SUBAPPLICATION RampLimitFS_TO_logiBUS_QDA_PWM_OPC (* Ein PWM-Kanal (0-100% Duty): VT-Zahlenfeld+Balkengrafik+6 Ramp-Tasten, physischer PWM-Ausgang, OPC-UA Publish/Subscribe (generisch, ein Kanal) *)
  (* Standard: 61499-2; Description: Copyright (c) 2026 Meisterschulen am Ostbahnhof This program and the accompanying materials are made available under the terms of the Eclipse Public License 2.0 which is available at https://www.eclipse.org/legal/epl-2.0/ SPDX-License-Identifier: EPL-2.0 *)
  (* Version 1.0, 2026-08-28, Franz Höpfinger, Meisterschulen am Ostbahnhof, initial API and implementation and/or initial documentation *)
  PACKAGE MyLib::sys;
  IMPORT isobus::UT::Q::const::IDs::ID_NULL;
  IMPORT logiBUS::io::DQ::logiBUS_DO;
  IMPORT logiBUS::io::DQ::logiBUS_DO_S;
  IMPORT isobus::UT::io::Button::ButtonActivationCode::BT_PRESSED_LATCHED;
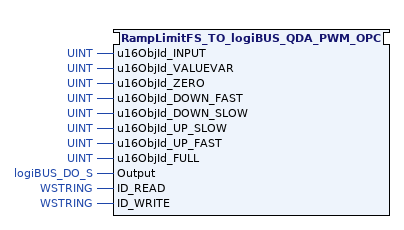
  VAR_INPUT
    u16ObjId_INPUT : UINT := ID_NULL; (* Object ID CInputNumber (Duty-Eingabe/-Anzeige, roh 0..64255 = 0.000-100.000%) *)
    u16ObjId_VALUEVAR : UINT := ID_NULL; (* Object ID CNumberVariable (Prozent 0-100, gemeinsam gebunden an Balkengrafik und CInputNumber-Anzeige) *)
    u16ObjId_ZERO : UINT := ID_NULL; (* Object ID Taste '0' (RampLimitFS.ZERO) *)
    u16ObjId_DOWN_FAST : UINT := ID_NULL; (* Object ID Taste '--' (RampLimitFS.DOWN_FAST, ~10%) *)
    u16ObjId_DOWN_SLOW : UINT := ID_NULL; (* Object ID Taste '-' (RampLimitFS.DOWN_SLOW, ~1%) *)
    u16ObjId_UP_SLOW : UINT := ID_NULL; (* Object ID Taste '+' (RampLimitFS.UP_SLOW, ~1%) *)
    u16ObjId_UP_FAST : UINT := ID_NULL; (* Object ID Taste '++' (RampLimitFS.UP_FAST, ~10%) *)
    u16ObjId_FULL : UINT := ID_NULL; (* Object ID Taste 'F' (RampLimitFS.FULL, 100%) *)
    Output : logiBUS::io::DQ::logiBUS_DO_S := logiBUS_DO::Invalid; (* Identify the PWM Output Output_Q1..Q12 *)
    ID_READ : WSTRING; (* Remote-Sollwert-Adresse (Prozent REAL, ACTION=SUBSCRIBE) *)
    ID_WRITE : WSTRING; (* Echo-Ruckmelde-Adresse (Prozent REAL, ACTION=PUBLISH) *)
  END_VAR
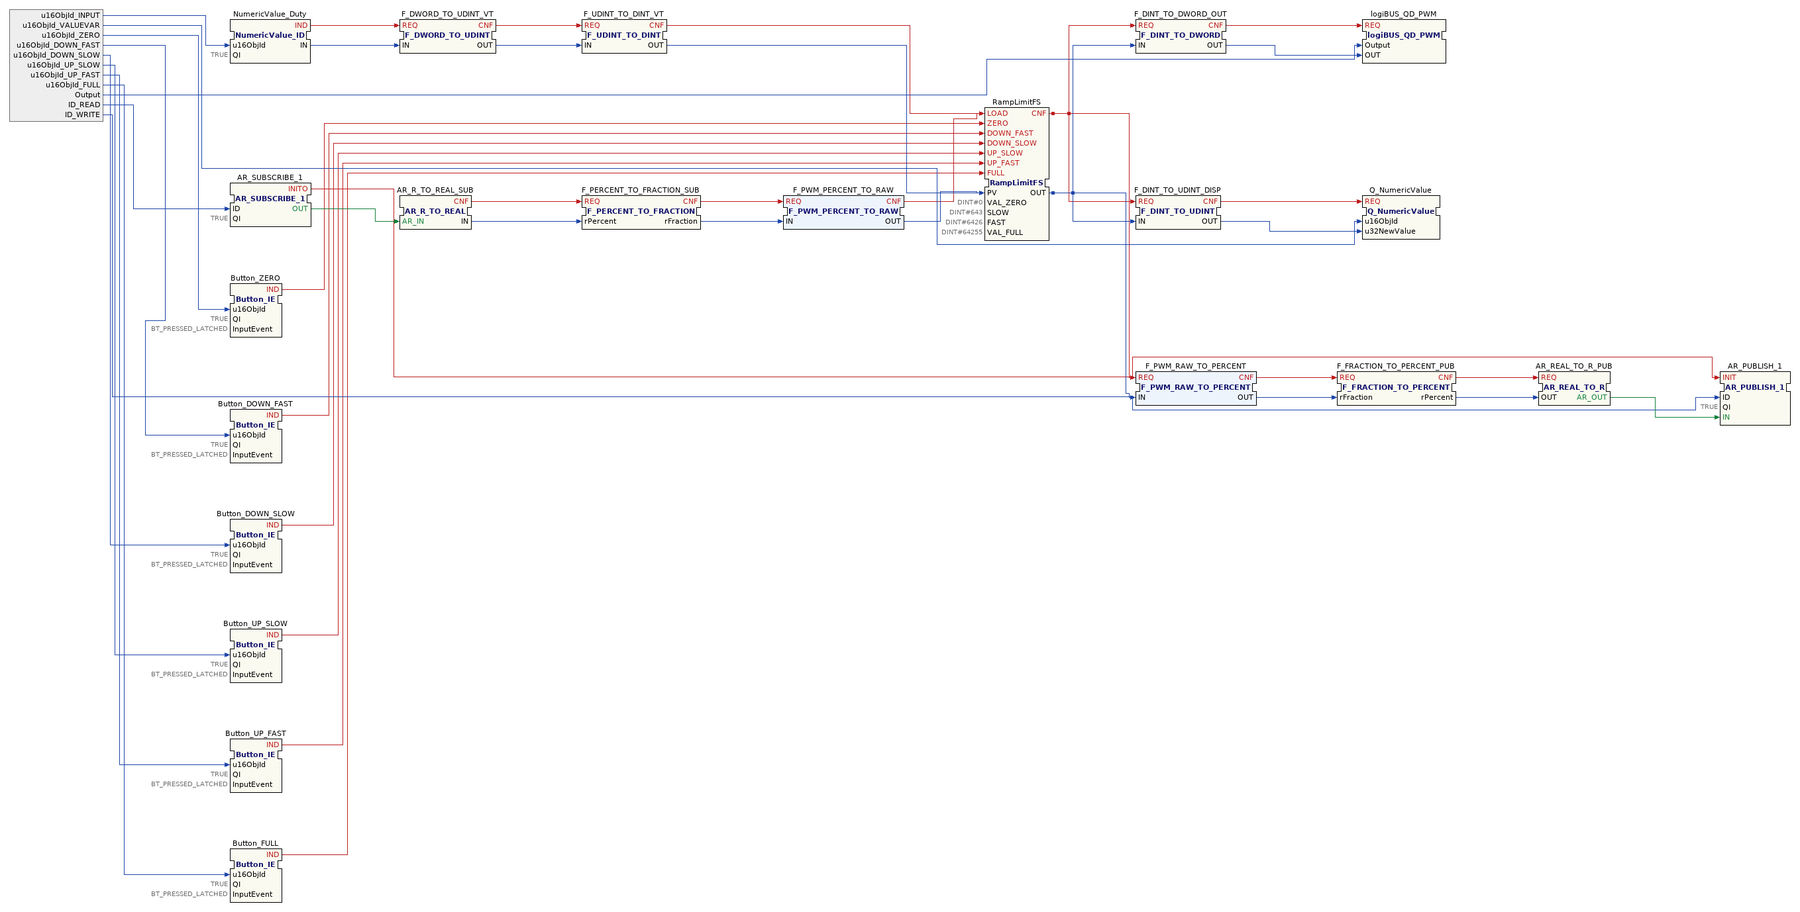
  FBS
    NumericValue_Duty : isobus::UT::io::NumericValue::NumericValue_ID(QI := TRUE);
    F_DWORD_TO_UDINT_VT : iec61131::conversion::F_DWORD_TO_UDINT;
    F_UDINT_TO_DINT_VT : iec61131::conversion::F_UDINT_TO_DINT;
    AR_SUBSCRIBE_1 : adapter::net::AR_SUBSCRIBE_1(QI := TRUE);
    AR_R_TO_REAL_SUB : adapter::conversion::unidirectional::AR_R_TO_REAL;
    F_PERCENT_TO_FRACTION_SUB : logiBUS::signalprocessing::fieldbus::F_PERCENT_TO_FRACTION;
    RampLimitFS : eclipse4diac::signalprocessing::RampLimitFS(VAL_ZERO := DINT#0, SLOW := DINT#643, FAST := DINT#6426, VAL_FULL := DINT#64255);
    Button_ZERO : isobus::UT::io::Button::Button_IE(QI := TRUE, InputEvent := BT_PRESSED_LATCHED);
    Button_DOWN_FAST : isobus::UT::io::Button::Button_IE(QI := TRUE, InputEvent := BT_PRESSED_LATCHED);
    Button_DOWN_SLOW : isobus::UT::io::Button::Button_IE(QI := TRUE, InputEvent := BT_PRESSED_LATCHED);
    Button_UP_SLOW : isobus::UT::io::Button::Button_IE(QI := TRUE, InputEvent := BT_PRESSED_LATCHED);
    Button_UP_FAST : isobus::UT::io::Button::Button_IE(QI := TRUE, InputEvent := BT_PRESSED_LATCHED);
    Button_FULL : isobus::UT::io::Button::Button_IE(QI := TRUE, InputEvent := BT_PRESSED_LATCHED);
    F_DINT_TO_DWORD_OUT : iec61131::conversion::F_DINT_TO_DWORD;
    logiBUS_QD_PWM : logiBUS::io::DQ::logiBUS_QD_PWM;
    F_DINT_TO_UDINT_DISP : iec61131::conversion::F_DINT_TO_UDINT;
    Q_NumericValue : isobus::UT::Q::Q_NumericValue;
    F_FRACTION_TO_PERCENT_PUB : logiBUS::signalprocessing::fieldbus::F_FRACTION_TO_PERCENT;
    AR_REAL_TO_R_PUB : adapter::conversion::unidirectional::AR_REAL_TO_R;
    AR_PUBLISH_1 : adapter::net::AR_PUBLISH_1(QI := TRUE);
  END_FBS
  SUBAPPS
    F_PWM_PERCENT_TO_RAW : MyLib::sys::F_PWM_PERCENT_TO_RAW;
    F_PWM_RAW_TO_PERCENT : MyLib::sys::F_PWM_RAW_TO_PERCENT;
  END_SUBAPPS
  EVENT_CONNECTIONS
    NumericValue_Duty.IND TO F_DWORD_TO_UDINT_VT.REQ;
    F_DWORD_TO_UDINT_VT.CNF TO F_UDINT_TO_DINT_VT.REQ;
    F_UDINT_TO_DINT_VT.CNF TO RampLimitFS.LOAD;
    AR_SUBSCRIBE_1.INITO TO AR_PUBLISH_1.INIT;
    AR_R_TO_REAL_SUB.CNF TO F_PERCENT_TO_FRACTION_SUB.REQ;
    F_PERCENT_TO_FRACTION_SUB.CNF TO F_PWM_PERCENT_TO_RAW.REQ;
    F_PWM_PERCENT_TO_RAW.CNF TO RampLimitFS.LOAD;
    Button_ZERO.IND TO RampLimitFS.ZERO;
    Button_DOWN_FAST.IND TO RampLimitFS.DOWN_FAST;
    Button_DOWN_SLOW.IND TO RampLimitFS.DOWN_SLOW;
    Button_UP_SLOW.IND TO RampLimitFS.UP_SLOW;
    Button_UP_FAST.IND TO RampLimitFS.UP_FAST;
    Button_FULL.IND TO RampLimitFS.FULL;
    RampLimitFS.CNF TO F_DINT_TO_DWORD_OUT.REQ;
    RampLimitFS.CNF TO F_DINT_TO_UDINT_DISP.REQ;
    RampLimitFS.CNF TO F_PWM_RAW_TO_PERCENT.REQ;
    F_DINT_TO_DWORD_OUT.CNF TO logiBUS_QD_PWM.REQ;
    F_DINT_TO_UDINT_DISP.CNF TO Q_NumericValue.REQ;
    F_PWM_RAW_TO_PERCENT.CNF TO F_FRACTION_TO_PERCENT_PUB.REQ;
    F_FRACTION_TO_PERCENT_PUB.CNF TO AR_REAL_TO_R_PUB.REQ;
  END_CONNECTIONS
  DATA_CONNECTIONS
    u16ObjId_INPUT TO NumericValue_Duty.u16ObjId;
    u16ObjId_VALUEVAR TO Q_NumericValue.u16ObjId;
    u16ObjId_ZERO TO Button_ZERO.u16ObjId;
    u16ObjId_DOWN_FAST TO Button_DOWN_FAST.u16ObjId;
    u16ObjId_DOWN_SLOW TO Button_DOWN_SLOW.u16ObjId;
    u16ObjId_UP_SLOW TO Button_UP_SLOW.u16ObjId;
    u16ObjId_UP_FAST TO Button_UP_FAST.u16ObjId;
    u16ObjId_FULL TO Button_FULL.u16ObjId;
    Output TO logiBUS_QD_PWM.Output;
    ID_READ TO AR_SUBSCRIBE_1.ID;
    ID_WRITE TO AR_PUBLISH_1.ID;
    NumericValue_Duty.IN TO F_DWORD_TO_UDINT_VT.IN;
    F_DWORD_TO_UDINT_VT.OUT TO F_UDINT_TO_DINT_VT.IN;
    F_UDINT_TO_DINT_VT.OUT TO RampLimitFS.PV;
    AR_R_TO_REAL_SUB.IN TO F_PERCENT_TO_FRACTION_SUB.rPercent;
    F_PERCENT_TO_FRACTION_SUB.rFraction TO F_PWM_PERCENT_TO_RAW.IN;
    F_PWM_PERCENT_TO_RAW.OUT TO RampLimitFS.PV;
    RampLimitFS.OUT TO F_DINT_TO_DWORD_OUT.IN;
    RampLimitFS.OUT TO F_DINT_TO_UDINT_DISP.IN;
    RampLimitFS.OUT TO F_PWM_RAW_TO_PERCENT.IN;
    F_DINT_TO_DWORD_OUT.OUT TO logiBUS_QD_PWM.OUT;
    F_DINT_TO_UDINT_DISP.OUT TO Q_NumericValue.u32NewValue;
    F_PWM_RAW_TO_PERCENT.OUT TO F_FRACTION_TO_PERCENT_PUB.rFraction;
    F_FRACTION_TO_PERCENT_PUB.rPercent TO AR_REAL_TO_R_PUB.OUT;
  END_CONNECTIONS
  ADAPTER_CONNECTIONS
    AR_SUBSCRIBE_1.OUT TO AR_R_TO_REAL_SUB.AR_IN;
    AR_REAL_TO_R_PUB.AR_OUT TO AR_PUBLISH_1.IN;
  END_CONNECTIONS
END_SUBAPPLICATION
